PROGRAM MAIN
VAR
	rInput: REAL;
END_VAR

// Control functions
//TemperatureControl();
ReactorTemperatureControl();
LevelControl();
PressureControl();
ReactorLevelControl();
// MATLAB functions
DataAcquisition();
// Persist set variables
VariablePersistent();
// Serial communications
SerialCommunicationHandler();

// Test CSharp


//Vanhat
(*//IO.bOutput := HMI.bContactor;
HMI.iTemperatureDisplayValue := IO.iInput/10;
//Temperature Control state
IF HMI.bTemperatureControlSwitch = 1 THEN
	HMI.sTemperatureControlState := 'AUTO';
END_IF
IF HMI.bTemperatureControlSwitch = 0 THEN
	HMI.sTemperatureControlState := 'MAN';
END_IF
//Level Control state
IF HMI.bLevelControlSwitch = 1 THEN
	HMI.sLevelControlState := 'AUTO';
END_IF
IF HMI.bLevelControlSwitch = 0 THEN
	HMI.sLevelControlState := 'MAN';
END_IF
//Level Valve state
IF IO.bReactorLu = 1 THEN
	HMI.sLevelValveState := 'CLOSE';
END_IF
IF IO.bReactorLu = 0 THEN
	HMI.sLevelValveState := 'OPEN';
END_IF*)

END_PROGRAM

(* stored: Version 1.1.0.1, ProductVersion 3.1.4024.9
   POU MAIN: Id {dec5b1ca-8e16-4f49-8efb-57a750654862}, SpecialFunc None *)
